// TwinCAT 3 PLC project PLC1
// ProgramVersion: 3.1.4026.23
// libraries:
//   Tc2_EtherCAT, * (Beckhoff Automation GmbH)
//   Tc2_Standard, * (Beckhoff Automation GmbH)
//   Tc2_System, * (Beckhoff Automation GmbH)
// project tree:
//   / Plc1Task.TcTTO
//   POUs/ F_ConsumeTime.TcPOU (not stored), PRG_PLC1.TcPOU
// real-time tasks:
//   TASK Plc1Task: cycle T#10ms, priority 10, ADS port 350
//   TASK Plc2Task: cycle T#10ms, priority 14, ADS port 351
//   TASK EcSlaveTask: cycle T#10ms, priority 3, ADS port 352
// I/O:
//   DEVICE EtherCAT Slave, AmsNetId 192.168.1.102.2.255
//   DEVICE EtherCAT Master, AmsNetId 192.168.1.102.4.1
//     Box 1 (CX5140 EtherCAT slave) [CX5140 EtherCAT slave]
// variable links:
//   (this object) <-> EtherCAT Master/Box 1 (CX5140 EtherCAT slave)
//     Plc1Task Inputs/PRG_PLC1.EncoderValue <-> IO Inputs/Sim Encoder
//     Plc2Task Inputs/PRG_PLC2.EncoderValue <-> IO Inputs/Sim Encoder
//   (this object) <-> EtherCAT Slave
//     PlcTask Outputs/MAIN.Counter <-> Outputs/Encoder Sim

CONFIGURATION PLC1
    RESOURCE PLC ON TwinCAT3
        TASK Plc1Task(INTERVAL := T#10ms, PRIORITY := 10);
        PROGRAM PRG_PLC1 WITH Plc1Task : PRG_PLC1;
    END_RESOURCE
END_CONFIGURATION

// ---- POUs/PRG_PLC1.TcPOU
PROGRAM PRG_PLC1
VAR
	EncoderValue AT %I* : UINT;
	Pos					: LREAL;
	ProcessingTime		:UDINT:=50;
END_VAR

F_ConsumeTime(ProcessingTime);

Pos:= UINT_TO_LREAL(EncoderValue)*100;

END_PROGRAM
